ABB RAPID module: Module1.mod

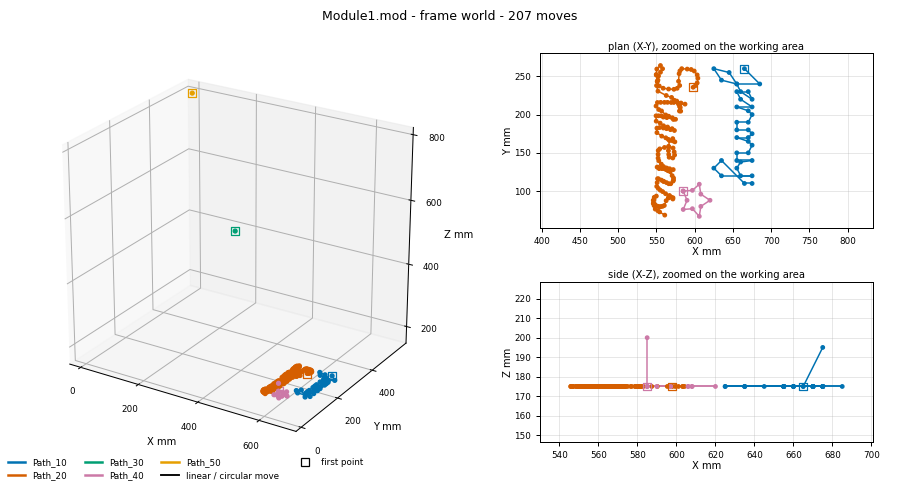
[picture p0: tool path of Module1.mod in frame world, 207 of 207 moves have a stored position in this frame; points joined in program order, loops and branches not executed]
MODULE Module1
    CONST robtarget Target_10:=[[45,210,0],[1,0,0,0],[0,0,-1,1],[9E+09,9E+09,9E+09,9E+09,9E+09,9E+09]];
    CONST robtarget Target_20:=[[25,190,0],[1,0,0,0],[0,0,-1,1],[9E+09,9E+09,9E+09,9E+09,9E+09,9E+09]];
    CONST robtarget Target_30:=[[55,190,0],[1,0,0,0],[0,0,-1,1],[9E+09,9E+09,9E+09,9E+09,9E+09,9E+09]];
    CONST robtarget Target_40:=[[75,195,0],[1,0,0,0],[0,0,-1,1],[9E+09,9E+09,9E+09,9E+09,9E+09,9E+09]];
    CONST robtarget Target_50:=[[85,210,0],[1,0,0,0],[0,0,-1,1],[9E+09,9E+09,9E+09,9E+09,9E+09,9E+09]];
    CONST robtarget Target_60:=[[65,205,0],[1,0,0,0],[0,0,-1,1],[9E+09,9E+09,9E+09,9E+09,9E+09,9E+09]];
    CONST robtarget Target_70:=[[55,190,0],[1,0,0,0],[0,0,-1,1],[9E+09,9E+09,9E+09,9E+09,9E+09,9E+09]];
    CONST robtarget Target_80:=[[50,180,0],[1,0,0,0],[0,0,-1,1],[9E+09,9E+09,9E+09,9E+09,9E+09,9E+09]];
    CONST robtarget Target_90:=[[35,170,0],[1,0,0,0],[0,0,-1,1],[9E+09,9E+09,9E+09,9E+09,9E+09,9E+09]];
    CONST robtarget Target_100:=[[40,180,0],[1,0,0,0],[0,0,-1,1],[9E+09,9E+09,9E+09,9E+09,9E+09,9E+09]];
    CONST robtarget Target_110:=[[55,180,0],[1,0,0,0],[0,0,-1,1],[9E+09,9E+09,9E+09,9E+09,9E+09,9E+09]];
    CONST robtarget Target_120:=[[50,170,0],[1,0,0,0],[0,0,-1,1],[9E+09,9E+09,9E+09,9E+09,9E+09,9E+09]];
    CONST robtarget Target_130:=[[35,160,0],[1,0,0,0],[0,0,-1,1],[9E+09,9E+09,9E+09,9E+09,9E+09,9E+09]];
    CONST robtarget Target_140:=[[55,160,0],[1,0,0,0],[0,0,-1,1],[9E+09,9E+09,9E+09,9E+09,9E+09,9E+09]];
    CONST robtarget Target_150:=[[40,155,0],[1,0,0,0],[0,0,-1,1],[9E+09,9E+09,9E+09,9E+09,9E+09,9E+09]];
    CONST robtarget Target_160:=[[35,150,0],[1,0,0,0],[0,0,-1,1],[9E+09,9E+09,9E+09,9E+09,9E+09,9E+09]];
    CONST robtarget Target_170:=[[40,140,0],[1,0,0,0],[0,0,-1,1],[9E+09,9E+09,9E+09,9E+09,9E+09,9E+09]];
    CONST robtarget Target_180:=[[55,140,0],[1,0,0,0],[0,0,-1,1],[9E+09,9E+09,9E+09,9E+09,9E+09,9E+09]];
    CONST robtarget Target_190:=[[55,130,0],[1,0,0,0],[0,0,-1,1],[9E+09,9E+09,9E+09,9E+09,9E+09,9E+09]];
    CONST robtarget Target_200:=[[40,130,0],[1,0,0,0],[0,0,-1,1],[9E+09,9E+09,9E+09,9E+09,9E+09,9E+09]];
    CONST robtarget Target_210:=[[35,125,0],[1,0,0,0],[0,0,-1,1],[9E+09,9E+09,9E+09,9E+09,9E+09,9E+09]];
    CONST robtarget Target_220:=[[40,120,0],[1,0,0,0],[0,0,-1,1],[9E+09,9E+09,9E+09,9E+09,9E+09,9E+09]];
    CONST robtarget Target_230:=[[55,120,0],[1,0,0,0],[0,0,-1,1],[9E+09,9E+09,9E+09,9E+09,9E+09,9E+09]];
    CONST robtarget Target_240:=[[40,115,0],[1,0,0,0],[0,0,-1,1],[9E+09,9E+09,9E+09,9E+09,9E+09,9E+09]];
    CONST robtarget Target_250:=[[35,110,0],[1,0,0,0],[0,0,-1,1],[9E+09,9E+09,9E+09,9E+09,9E+09,9E+09]];
    CONST robtarget Target_260:=[[40,100,0],[1,0,0,0],[0,0,-1,1],[9E+09,9E+09,9E+09,9E+09,9E+09,9E+09]];
    CONST robtarget Target_270:=[[55,100,0],[1,0,0,0],[0,0,-1,1],[9E+09,9E+09,9E+09,9E+09,9E+09,9E+09]];
    CONST robtarget Target_280:=[[55,90,0],[1,0,0,0],[0,0,-1,1],[9E+09,9E+09,9E+09,9E+09,9E+09,9E+09]];
    CONST robtarget Target_290:=[[35,90,0],[1,0,0,0],[0,0,-1,1],[9E+09,9E+09,9E+09,9E+09,9E+09,9E+09]];
    CONST robtarget Target_300:=[[50,88,0],[1,0,0,0],[0,0,-1,1],[9E+09,9E+09,9E+09,9E+09,9E+09,9E+09]];
    CONST robtarget Target_310:=[[55,80,0],[1,0,0,0],[0,0,-1,1],[9E+09,9E+09,9E+09,9E+09,9E+09,9E+09]];
    CONST robtarget Target_320:=[[50,70,0],[1,0,0,0],[0,0,-1,1],[9E+09,9E+09,9E+09,9E+09,9E+09,9E+09]];
    CONST robtarget Target_330:=[[35,70,0],[1,0,0,0],[0,0,-1,1],[9E+09,9E+09,9E+09,9E+09,9E+09,9E+09]];
    CONST robtarget Target_340:=[[75,70,0],[1,0,0,0],[0,0,-1,1],[9E+09,9E+09,9E+09,9E+09,9E+09,9E+09]];
    CONST robtarget Target_350:=[[85,80,0],[1,0,0,0],[0,0,-1,1],[9E+09,9E+09,9E+09,9E+09,9E+09,9E+09]];
    CONST robtarget Target_360:=[[75,90,0],[1,0,0,0],[0,0,-1,1],[9E+09,9E+09,9E+09,9E+09,9E+09,9E+09]];
    CONST robtarget Target_370:=[[45,60,0],[1,0,0,0],[0,0,-1,1],[9E+09,9E+09,9E+09,9E+09,9E+09,9E+09]];
    CONST robtarget Target_390:=[[108.942,187.897,0],[1,0,0,0],[0,0,-1,1],[9E+09,9E+09,9E+09,9E+09,9E+09,9E+09]];
    CONST robtarget Target_400:=[[106.749,191.385,0],[1,0,0,0],[0,0,-1,1],[9E+09,9E+09,9E+09,9E+09,9E+09,9E+09]];
    CONST robtarget Target_380:=[[112.054,185.689,0],[1,0,0,0],[0,0,-1,1],[9E+09,9E+09,9E+09,9E+09,9E+09,9E+09]];
    CONST robtarget Target_410:=[[105.843,197.618,0],[1,0,0,0],[0,0,-1,1],[9E+09,9E+09,9E+09,9E+09,9E+09,9E+09]];
    CONST robtarget Target_420:=[[106.766,201.829,0],[1,0,0,0],[0,0,-1,1],[9E+09,9E+09,9E+09,9E+09,9E+09,9E+09]];
    CONST robtarget Target_430:=[[110.623,206.946,0],[1,0,0,0],[0,0,-1,1],[9E+09,9E+09,9E+09,9E+09,9E+09,9E+09]];
    CONST robtarget Target_440:=[[114.657,208.948,0],[1,0,0,0],[0,0,-1,1],[9E+09,9E+09,9E+09,9E+09,9E+09,9E+09]];
    CONST robtarget Target_450:=[[119.787,209.479,0],[1,0,0,0],[0,0,-1,1],[9E+09,9E+09,9E+09,9E+09,9E+09,9E+09]];
    CONST robtarget Target_460:=[[126.931,210.004,0],[1,0,0,0],[0,0,-1,1],[9E+09,9E+09,9E+09,9E+09,9E+09,9E+09]];
    CONST robtarget Target_470:=[[129.306,207.065,0],[1,0,0,0],[0,0,-1,1],[9E+09,9E+09,9E+09,9E+09,9E+09,9E+09]];
    CONST robtarget Target_480:=[[130.399,203.399,0],[1,0,0,0],[0,0,-1,1],[9E+09,9E+09,9E+09,9E+09,9E+09,9E+09]];
    CONST robtarget Target_490:=[[131.115,193.507,0],[1,0,0,0],[0,0,-1,1],[9E+09,9E+09,9E+09,9E+09,9E+09,9E+09]];
    CONST robtarget Target_500:=[[129.641,188.017,0],[1,0,0,0],[0,0,-1,1],[9E+09,9E+09,9E+09,9E+09,9E+09,9E+09]];
    CONST robtarget Target_510:=[[132.931,184.344,0],[1,0,0,0],[0,0,-1,1],[9E+09,9E+09,9E+09,9E+09,9E+09,9E+09]];
    CONST robtarget Target_520:=[[137.139,183.05,0],[1,0,0,0],[0,0,-1,1],[9E+09,9E+09,9E+09,9E+09,9E+09,9E+09]];
    CONST robtarget Target_530:=[[144.094,183.396,0],[1,0,0,0],[0,0,-1,1],[9E+09,9E+09,9E+09,9E+09,9E+09,9E+09]];
    CONST robtarget Target_540:=[[151.231,184.473,0],[1,0,0,0],[0,0,-1,1],[9E+09,9E+09,9E+09,9E+09,9E+09,9E+09]];
    CONST robtarget Target_550:=[[156.358,187.386,0],[1,0,0,0],[0,0,-1,1],[9E+09,9E+09,9E+09,9E+09,9E+09,9E+09]];
    CONST robtarget Target_560:=[[158.928,193.236,0],[1,0,0,0],[0,0,-1,1],[9E+09,9E+09,9E+09,9E+09,9E+09,9E+09]];
    CONST robtarget Target_570:=[[158.929,193.602,0],[1,0,0,0],[0,0,-1,1],[9E+09,9E+09,9E+09,9E+09,9E+09,9E+09]];
    CONST robtarget Target_580:=[[160.222,201.651,0],[1,0,0,0],[0,0,-1,1],[9E+09,9E+09,9E+09,9E+09,9E+09,9E+09]];
    CONST robtarget Target_590:=[[160.223,202.383,0],[1,0,0,0],[0,0,-1,1],[9E+09,9E+09,9E+09,9E+09,9E+09,9E+09]];
    CONST robtarget Target_600:=[[159.504,209.524,0],[1,0,0,0],[0,0,-1,1],[9E+09,9E+09,9E+09,9E+09,9E+09,9E+09]];
    CONST robtarget Target_610:=[[154.756,214.117,0],[1,0,0,0],[0,0,-1,1],[9E+09,9E+09,9E+09,9E+09,9E+09,9E+09]];
    CONST robtarget Target_620:=[[152.005,209.916,0],[1,0,0,0],[0,0,-1,1],[9E+09,9E+09,9E+09,9E+09,9E+09,9E+09]];
    CONST robtarget Target_630:=[[154.741,205.33,0],[1,0,0,0],[0,0,-1,1],[9E+09,9E+09,9E+09,9E+09,9E+09,9E+09]];
    CONST robtarget Target_640:=[[157.294,200.379,0],[1,0,0,0],[0,0,-1,1],[9E+09,9E+09,9E+09,9E+09,9E+09,9E+09]];
    CONST robtarget Target_650:=[[158.017,195.069,0],[1,0,0,0],[0,0,-1,1],[9E+09,9E+09,9E+09,9E+09,9E+09,9E+09]];
    CONST robtarget Target_660:=[[159.834,187.925,0],[1,0,0,0],[0,0,-1,1],[9E+09,9E+09,9E+09,9E+09,9E+09,9E+09]];
    CONST robtarget Target_670:=[[157.993,180.609,0],[1,0,0,0],[0,0,-1,1],[9E+09,9E+09,9E+09,9E+09,9E+09,9E+09]];
    CONST robtarget Target_680:=[[147.191,174.965,0],[1,0,0,0],[0,0,-1,1],[9E+09,9E+09,9E+09,9E+09,9E+09,9E+09]];
    CONST robtarget Target_690:=[[140.233,172.421,0],[1,0,0,0],[0,0,-1,1],[9E+09,9E+09,9E+09,9E+09,9E+09,9E+09]];
    CONST robtarget Target_700:=[[136.749,168.768,0],[1,0,0,0],[0,0,-1,1],[9E+09,9E+09,9E+09,9E+09,9E+09,9E+09]];
    CONST robtarget Target_710:=[[133.452,167.678,0],[1,0,0,0],[0,0,-1,1],[9E+09,9E+09,9E+09,9E+09,9E+09,9E+09]];
    CONST robtarget Target_720:=[[127.955,165.128,0],[1,0,0,0],[0,0,-1,1],[9E+09,9E+09,9E+09,9E+09,9E+09,9E+09]];
    CONST robtarget Target_730:=[[122.642,163.677,0],[1,0,0,0],[0,0,-1,1],[9E+09,9E+09,9E+09,9E+09,9E+09,9E+09]];
    CONST robtarget Target_740:=[[128.504,164.578,0],[1,0,0,0],[0,0,-1,1],[9E+09,9E+09,9E+09,9E+09,9E+09,9E+09]];
    CONST robtarget Target_750:=[[129.779,160.545,0],[1,0,0,0],[0,0,-1,1],[9E+09,9E+09,9E+09,9E+09,9E+09,9E+09]];
    CONST robtarget Target_760:=[[129.952,154.684,0],[1,0,0,0],[0,0,-1,1],[9E+09,9E+09,9E+09,9E+09,9E+09,9E+09]];
    CONST robtarget Target_770:=[[128.304,154.505,0],[1,0,0,0],[0,0,-1,1],[9E+09,9E+09,9E+09,9E+09,9E+09,9E+09]];
    CONST robtarget Target_780:=[[128.861,159.265,0],[1,0,0,0],[0,0,-1,1],[9E+09,9E+09,9E+09,9E+09,9E+09,9E+09]];
    CONST robtarget Target_790:=[[131.249,163.838,0],[1,0,0,0],[0,0,-1,1],[9E+09,9E+09,9E+09,9E+09,9E+09,9E+09]];
    CONST robtarget Target_800:=[[137.293,165.837,0],[1,0,0,0],[0,0,-1,1],[9E+09,9E+09,9E+09,9E+09,9E+09,9E+09]];
    CONST robtarget Target_810:=[[140.771,165.828,0],[1,0,0,0],[0,0,-1,1],[9E+09,9E+09,9E+09,9E+09,9E+09,9E+09]];
    CONST robtarget Target_820:=[[145.529,165.998,0],[1,0,0,0],[0,0,-1,1],[9E+09,9E+09,9E+09,9E+09,9E+09,9E+09]];
    CONST robtarget Target_830:=[[149.554,165.988,0],[1,0,0,0],[0,0,-1,1],[9E+09,9E+09,9E+09,9E+09,9E+09,9E+09]];
    CONST robtarget Target_840:=[[154.494,165.975,0],[1,0,0,0],[0,0,-1,1],[9E+09,9E+09,9E+09,9E+09,9E+09,9E+09]];
    CONST robtarget Target_850:=[[158.7,165.781,0],[1,0,0,0],[0,0,-1,1],[9E+09,9E+09,9E+09,9E+09,9E+09,9E+09]];
    CONST robtarget Target_860:=[[160.521,161.2,0],[1,0,0,0],[0,0,-1,1],[9E+09,9E+09,9E+09,9E+09,9E+09,9E+09]];
    CONST robtarget Target_870:=[[157.039,156.633,0],[1,0,0,0],[0,0,-1,1],[9E+09,9E+09,9E+09,9E+09,9E+09,9E+09]];
    CONST robtarget Target_880:=[[153.378,154.811,0],[1,0,0,0],[0,0,-1,1],[9E+09,9E+09,9E+09,9E+09,9E+09,9E+09]];
    CONST robtarget Target_890:=[[147.881,149.515,0],[1,0,0,0],[0,0,-1,1],[9E+09,9E+09,9E+09,9E+09,9E+09,9E+09]];
    CONST robtarget Target_900:=[[144.035,147.876,0],[1,0,0,0],[0,0,-1,1],[9E+09,9E+09,9E+09,9E+09,9E+09,9E+09]];
    CONST robtarget Target_910:=[[139.274,145.873,0],[1,0,0,0],[0,0,-1,1],[9E+09,9E+09,9E+09,9E+09,9E+09,9E+09]];
    CONST robtarget Target_920:=[[135.061,143.868,0],[1,0,0,0],[0,0,-1,1],[9E+09,9E+09,9E+09,9E+09,9E+09,9E+09]];
    CONST robtarget Target_930:=[[137.806,143.679,0],[1,0,0,0],[0,0,-1,1],[9E+09,9E+09,9E+09,9E+09,9E+09,9E+09]];
    CONST robtarget Target_940:=[[146.411,146.04,0],[1,0,0,0],[0,0,-1,1],[9E+09,9E+09,9E+09,9E+09,9E+09,9E+09]];
    CONST robtarget Target_960:=[[153.733,148.403,0],[1,0,0,0],[0,0,-1,1],[9E+09,9E+09,9E+09,9E+09,9E+09,9E+09]];
    CONST robtarget Target_970:=[[157.391,148.395,0],[1,0,0,0],[0,0,-1,1],[9E+09,9E+09,9E+09,9E+09,9E+09,9E+09]];
    CONST robtarget Target_980:=[[160.5,148.388,0],[1,0,0,0],[0,0,-1,1],[9E+09,9E+09,9E+09,9E+09,9E+09,9E+09]];
    CONST robtarget Target_990:=[[160.306,141.433,0],[1,0,0,0],[0,0,-1,1],[9E+09,9E+09,9E+09,9E+09,9E+09,9E+09]];
    CONST robtarget Target_1000:=[[155.181,138.881,0],[1,0,0,0],[0,0,-1,1],[9E+09,9E+09,9E+09,9E+09,9E+09,9E+09]];
    CONST robtarget Target_1010:=[[150.785,135.412,0],[1,0,0,0],[0,0,-1,1],[9E+09,9E+09,9E+09,9E+09,9E+09,9E+09]];
    CONST robtarget Target_1020:=[[145.476,133.775,0],[1,0,0,0],[0,0,-1,1],[9E+09,9E+09,9E+09,9E+09,9E+09,9E+09]];
    CONST robtarget Target_1030:=[[139.616,131.59,0],[1,0,0,0],[0,0,-1,1],[9E+09,9E+09,9E+09,9E+09,9E+09,9E+09]];
    CONST robtarget Target_1040:=[[136.501,129.215,0],[1,0,0,0],[0,0,-1,1],[9E+09,9E+09,9E+09,9E+09,9E+09,9E+09]];
    CONST robtarget Target_1050:=[[141.627,130.304,0],[1,0,0,0],[0,0,-1,1],[9E+09,9E+09,9E+09,9E+09,9E+09,9E+09]];
    CONST robtarget Target_1060:=[[146.753,131.576,0],[1,0,0,0],[0,0,-1,1],[9E+09,9E+09,9E+09,9E+09,9E+09,9E+09]];
    CONST robtarget Target_1070:=[[150.963,132.483,0],[1,0,0,0],[0,0,-1,1],[9E+09,9E+09,9E+09,9E+09,9E+09,9E+09]];
    CONST robtarget Target_1080:=[[155.903,133.022,0],[1,0,0,0],[0,0,-1,1],[9E+09,9E+09,9E+09,9E+09,9E+09,9E+09]];
    CONST robtarget Target_1090:=[[159.376,132.284,0],[1,0,0,0],[0,0,-1,1],[9E+09,9E+09,9E+09,9E+09,9E+09,9E+09]];
    CONST robtarget Target_1100:=[[159.367,126.426,0],[1,0,0,0],[0,0,-1,1],[9E+09,9E+09,9E+09,9E+09,9E+09,9E+09]];
    CONST robtarget Target_1110:=[[153.14,121.861,0],[1,0,0,0],[0,0,-1,1],[9E+09,9E+09,9E+09,9E+09,9E+09,9E+09]];
    CONST robtarget Target_1120:=[[147.831,119.674,0],[1,0,0,0],[0,0,-1,1],[9E+09,9E+09,9E+09,9E+09,9E+09,9E+09]];
    CONST robtarget Target_1130:=[[144.535,117.665,0],[1,0,0,0],[0,0,-1,1],[9E+09,9E+09,9E+09,9E+09,9E+09,9E+09]];
    CONST robtarget Target_1140:=[[138.675,115.661,0],[1,0,0,0],[0,0,-1,1],[9E+09,9E+09,9E+09,9E+09,9E+09,9E+09]];
    CONST robtarget Target_1150:=[[135.927,114.383,0],[1,0,0,0],[0,0,-1,1],[9E+09,9E+09,9E+09,9E+09,9E+09,9E+09]];
    CONST robtarget Target_1160:=[[138.68,118.591,0],[1,0,0,0],[0,0,-1,1],[9E+09,9E+09,9E+09,9E+09,9E+09,9E+09]];
    CONST robtarget Target_1170:=[[142.885,116.02,0],[1,0,0,0],[0,0,-1,1],[9E+09,9E+09,9E+09,9E+09,9E+09,9E+09]];
    CONST robtarget Target_1180:=[[144.154,108.511,0],[1,0,0,0],[0,0,-1,1],[9E+09,9E+09,9E+09,9E+09,9E+09,9E+09]];
    CONST robtarget Target_1190:=[[144.327,102.835,0],[1,0,0,0],[0,0,-1,1],[9E+09,9E+09,9E+09,9E+09,9E+09,9E+09]];
    CONST robtarget Target_1200:=[[143.953,97.892,0],[1,0,0,0],[0,0,-1,1],[9E+09,9E+09,9E+09,9E+09,9E+09,9E+09]];
    CONST robtarget Target_1210:=[[143.398,94.231,0],[1,0,0,0],[0,0,-1,1],[9E+09,9E+09,9E+09,9E+09,9E+09,9E+09]];
    CONST robtarget Target_1220:=[[138.638,93.321,0],[1,0,0,0],[0,0,-1,1],[9E+09,9E+09,9E+09,9E+09,9E+09,9E+09]];
    CONST robtarget Target_1230:=[[136.265,97.17,0],[1,0,0,0],[0,0,-1,1],[9E+09,9E+09,9E+09,9E+09,9E+09,9E+09]];
    CONST robtarget Target_1240:=[[136.821,101.198,0],[1,0,0,0],[0,0,-1,1],[9E+09,9E+09,9E+09,9E+09,9E+09,9E+09]];
    CONST robtarget Target_1250:=[[138.294,106.323,0],[1,0,0,0],[0,0,-1,1],[9E+09,9E+09,9E+09,9E+09,9E+09,9E+09]];
    CONST robtarget Target_1260:=[[143.786,107.597,0],[1,0,0,0],[0,0,-1,1],[9E+09,9E+09,9E+09,9E+09,9E+09,9E+09]];
    CONST robtarget Target_1270:=[[149.457,107.039,0],[1,0,0,0],[0,0,-1,1],[9E+09,9E+09,9E+09,9E+09,9E+09,9E+09]];
    CONST robtarget Target_1280:=[[155.674,105.2,0],[1,0,0,0],[0,0,-1,1],[9E+09,9E+09,9E+09,9E+09,9E+09,9E+09]];
    CONST robtarget Target_1290:=[[157.682,103,0],[1,0,0,0],[0,0,-1,1],[9E+09,9E+09,9E+09,9E+09,9E+09,9E+09]];
    CONST robtarget Target_1300:=[[157.857,98.058,0],[1,0,0,0],[0,0,-1,1],[9E+09,9E+09,9E+09,9E+09,9E+09,9E+09]];
    CONST robtarget Target_1310:=[[157.849,93.116,0],[1,0,0,0],[0,0,-1,1],[9E+09,9E+09,9E+09,9E+09,9E+09,9E+09]];
    CONST robtarget Target_1320:=[[156.928,89.639,0],[1,0,0,0],[0,0,-1,1],[9E+09,9E+09,9E+09,9E+09,9E+09,9E+09]];
    CONST robtarget Target_1330:=[[153.629,85.25,0],[1,0,0,0],[0,0,-1,1],[9E+09,9E+09,9E+09,9E+09,9E+09,9E+09]];
    CONST robtarget Target_1340:=[[150.88,82.14,0],[1,0,0,0],[0,0,-1,1],[9E+09,9E+09,9E+09,9E+09,9E+09,9E+09]];
    CONST robtarget Target_1350:=[[147.035,80.313,0],[1,0,0,0],[0,0,-1,1],[9E+09,9E+09,9E+09,9E+09,9E+09,9E+09]];
    CONST robtarget Target_1360:=[[142.824,79.218,0],[1,0,0,0],[0,0,-1,1],[9E+09,9E+09,9E+09,9E+09,9E+09,9E+09]];
    CONST robtarget Target_1370:=[[138.064,78.124,0],[1,0,0,0],[0,0,-1,1],[9E+09,9E+09,9E+09,9E+09,9E+09,9E+09]];
    CONST robtarget Target_1380:=[[141.907,77.754,0],[1,0,0,0],[0,0,-1,1],[9E+09,9E+09,9E+09,9E+09,9E+09,9E+09]];
    CONST robtarget Target_1390:=[[145.752,79.216,0],[1,0,0,0],[0,0,-1,1],[9E+09,9E+09,9E+09,9E+09,9E+09,9E+09]];
    CONST robtarget Target_1400:=[[149.412,79.396,0],[1,0,0,0],[0,0,-1,1],[9E+09,9E+09,9E+09,9E+09,9E+09,9E+09]];
    CONST robtarget Target_1410:=[[154.17,80.856,0],[1,0,0,0],[0,0,-1,1],[9E+09,9E+09,9E+09,9E+09,9E+09,9E+09]];
    CONST robtarget Target_1420:=[[158.012,81.218,0],[1,0,0,0],[0,0,-1,1],[9E+09,9E+09,9E+09,9E+09,9E+09,9E+09]];
    CONST robtarget Target_1430:=[[159.11,81.4,0],[1,0,0,0],[0,0,-1,1],[9E+09,9E+09,9E+09,9E+09,9E+09,9E+09]];
    CONST robtarget Target_1440:=[[156.546,79.389,0],[1,0,0,0],[0,0,-1,1],[9E+09,9E+09,9E+09,9E+09,9E+09,9E+09]];
    CONST robtarget Target_1450:=[[152.888,79.392,0],[1,0,0,0],[0,0,-1,1],[9E+09,9E+09,9E+09,9E+09,9E+09,9E+09]];
    CONST robtarget Target_1460:=[[150.327,79.578,0],[1,0,0,0],[0,0,-1,1],[9E+09,9E+09,9E+09,9E+09,9E+09,9E+09]];
    CONST robtarget Target_1470:=[[147.58,78.116,0],[1,0,0,0],[0,0,-1,1],[9E+09,9E+09,9E+09,9E+09,9E+09,9E+09]];
    CONST robtarget Target_1480:=[[145.016,76.653,0],[1,0,0,0],[0,0,-1,1],[9E+09,9E+09,9E+09,9E+09,9E+09,9E+09]];
    CONST robtarget Target_1490:=[[142.086,75.374,0],[1,0,0,0],[0,0,-1,1],[9E+09,9E+09,9E+09,9E+09,9E+09,9E+09]];
    CONST robtarget Target_1500:=[[139.515,70.249,0],[1,0,0,0],[0,0,-1,1],[9E+09,9E+09,9E+09,9E+09,9E+09,9E+09]];
    CONST robtarget Target_1510:=[[137.68,67.137,0],[1,0,0,0],[0,0,-1,1],[9E+09,9E+09,9E+09,9E+09,9E+09,9E+09]];
    CONST robtarget Target_1520:=[[137.676,64.574,0],[1,0,0,0],[0,0,-1,1],[9E+09,9E+09,9E+09,9E+09,9E+09,9E+09]];
    CONST robtarget Target_1530:=[[138.222,63.109,0],[1,0,0,0],[0,0,-1,1],[9E+09,9E+09,9E+09,9E+09,9E+09,9E+09]];
    CONST robtarget Target_1540:=[[141.328,59.628,0],[1,0,0,0],[0,0,-1,1],[9E+09,9E+09,9E+09,9E+09,9E+09,9E+09]];
    CONST robtarget Target_1550:=[[143.89,59.627,0],[1,0,0,0],[0,0,-1,1],[9E+09,9E+09,9E+09,9E+09,9E+09,9E+09]];
    CONST robtarget Target_1560:=[[146.82,61.09,0],[1,0,0,0],[0,0,-1,1],[9E+09,9E+09,9E+09,9E+09,9E+09,9E+09]];
    CONST robtarget Target_1570:=[[150.299,62.553,0],[1,0,0,0],[0,0,-1,1],[9E+09,9E+09,9E+09,9E+09,9E+09,9E+09]];
    CONST robtarget Target_1580:=[[151.031,62.918,0],[1,0,0,0],[0,0,-1,1],[9E+09,9E+09,9E+09,9E+09,9E+09,9E+09]];
    CONST robtarget Target_1590:=[[153.594,64.381,0],[1,0,0,0],[0,0,-1,1],[9E+09,9E+09,9E+09,9E+09,9E+09,9E+09]];
    CONST robtarget Target_1600:=[[157.255,66.026,0],[1,0,0,0],[0,0,-1,1],[9E+09,9E+09,9E+09,9E+09,9E+09,9E+09]];
    CONST robtarget Target_1610:=[[158.536,66.209,0],[1,0,0,0],[0,0,-1,1],[9E+09,9E+09,9E+09,9E+09,9E+09,9E+09]];
    CONST robtarget Target_1620:=[[159.076,61.083,0],[1,0,0,0],[0,0,-1,1],[9E+09,9E+09,9E+09,9E+09,9E+09,9E+09]];
    CONST robtarget Target_1630:=[[159.617,56.141,0],[1,0,0,0],[0,0,-1,1],[9E+09,9E+09,9E+09,9E+09,9E+09,9E+09]];
    CONST robtarget Target_1640:=[[157.601,53.58,0],[1,0,0,0],[0,0,-1,1],[9E+09,9E+09,9E+09,9E+09,9E+09,9E+09]];
    CONST robtarget Target_1650:=[[155.036,51.201,0],[1,0,0,0],[0,0,-1,1],[9E+09,9E+09,9E+09,9E+09,9E+09,9E+09]];
    CONST robtarget Target_1660:=[[151.923,49.371,0],[1,0,0,0],[0,0,-1,1],[9E+09,9E+09,9E+09,9E+09,9E+09,9E+09]];
    CONST robtarget Target_1670:=[[148.077,46.626,0],[1,0,0,0],[0,0,-1,1],[9E+09,9E+09,9E+09,9E+09,9E+09,9E+09]];
    CONST robtarget Target_1680:=[[142.95,44.247,0],[1,0,0,0],[0,0,-1,1],[9E+09,9E+09,9E+09,9E+09,9E+09,9E+09]];
    CONST robtarget Target_1690:=[[138.55,39.67,0],[1,0,0,0],[0,0,-1,1],[9E+09,9E+09,9E+09,9E+09,9E+09,9E+09]];
    CONST robtarget Target_1700:=[[138.369,41.318,0],[1,0,0,0],[0,0,-1,1],[9E+09,9E+09,9E+09,9E+09,9E+09,9E+09]];
    CONST robtarget Target_1710:=[[140.567,42.05,0],[1,0,0,0],[0,0,-1,1],[9E+09,9E+09,9E+09,9E+09,9E+09,9E+09]];
    CONST robtarget Target_1720:=[[143.13,42.599,0],[1,0,0,0],[0,0,-1,1],[9E+09,9E+09,9E+09,9E+09,9E+09,9E+09]];
    CONST robtarget Target_1730:=[[144.226,41.501,0],[1,0,0,0],[0,0,-1,1],[9E+09,9E+09,9E+09,9E+09,9E+09,9E+09]];
    CONST robtarget Target_1740:=[[144.408,40.951,0],[1,0,0,0],[0,0,-1,1],[9E+09,9E+09,9E+09,9E+09,9E+09,9E+09]];
    CONST robtarget Target_1750:=[[147.33,37.473,0],[1,0,0,0],[0,0,-1,1],[9E+09,9E+09,9E+09,9E+09,9E+09,9E+09]];
    CONST robtarget Target_1760:=[[149.698,31.248,0],[1,0,0,0],[0,0,-1,1],[9E+09,9E+09,9E+09,9E+09,9E+09,9E+09]];
    CONST robtarget Target_1770:=[[151.892,30.15,0],[1,0,0,0],[0,0,-1,1],[9E+09,9E+09,9E+09,9E+09,9E+09,9E+09]];
    CONST robtarget Target_1780:=[[154.086,29.784,0],[1,0,0,0],[0,0,-1,1],[9E+09,9E+09,9E+09,9E+09,9E+09,9E+09]];
    CONST robtarget Target_1790:=[[156.098,29.601,0],[1,0,0,0],[0,0,-1,1],[9E+09,9E+09,9E+09,9E+09,9E+09,9E+09]];
    CONST robtarget Target_1800:=[[158.111,30.15,0],[1,0,0,0],[0,0,-1,1],[9E+09,9E+09,9E+09,9E+09,9E+09,9E+09]];
    CONST robtarget Target_1810:=[[161.405,31.981,0],[1,0,0,0],[0,0,-1,1],[9E+09,9E+09,9E+09,9E+09,9E+09,9E+09]];
    CONST robtarget Target_1820:=[[164.151,33.811,0],[1,0,0,0],[0,0,-1,1],[9E+09,9E+09,9E+09,9E+09,9E+09,9E+09]];
    CONST robtarget Target_1830:=[[164.158,37.838,0],[1,0,0,0],[0,0,-1,1],[9E+09,9E+09,9E+09,9E+09,9E+09,9E+09]];
    CONST robtarget Target_1840:=[[162.885,41.864,0],[1,0,0,0],[0,0,-1,1],[9E+09,9E+09,9E+09,9E+09,9E+09,9E+09]];
    CONST robtarget Target_1850:=[[160.144,43.512,0],[1,0,0,0],[0,0,-1,1],[9E+09,9E+09,9E+09,9E+09,9E+09,9E+09]];
    CONST robtarget Target_1860:=[[163.245,38.753,0],[1,0,0,0],[0,0,-1,1],[9E+09,9E+09,9E+09,9E+09,9E+09,9E+09]];
    CONST robtarget Target_1870:=[[163.604,34.543,0],[1,0,0,0],[0,0,-1,1],[9E+09,9E+09,9E+09,9E+09,9E+09,9E+09]];
    CONST robtarget Target_1880:=[[163.05,31.066,0],[1,0,0,0],[0,0,-1,1],[9E+09,9E+09,9E+09,9E+09,9E+09,9E+09]];
    CONST robtarget Target_1890:=[[161.579,26.49,0],[1,0,0,0],[0,0,-1,1],[9E+09,9E+09,9E+09,9E+09,9E+09,9E+09]];
    CONST robtarget Target_1900:=[[158.101,24.293,0],[1,0,0,0],[0,0,-1,1],[9E+09,9E+09,9E+09,9E+09,9E+09,9E+09]];
    CONST robtarget Target_1910:=[[155.904,22.828,0],[1,0,0,0],[0,0,-1,1],[9E+09,9E+09,9E+09,9E+09,9E+09,9E+09]];
    CONST robtarget Target_1920:=[[149.128,18.616,0],[1,0,0,0],[0,0,-1,1],[9E+09,9E+09,9E+09,9E+09,9E+09,9E+09]];
    CONST robtarget Target_950:=[[150.986,146.762,0],[1,0,0,0],[0,0,-1,1],[9E+09,9E+09,9E+09,9E+09,9E+09,9E+09]];
    CONST robtarget Target_Home:=[[506.291651246,0,679.5],[0.5,0,0.866025404,0],[0,0,-1,1],[9E+09,9E+09,9E+09,9E+09,9E+09,9E+09]];
    CONST robtarget Target_Up_first:=[[35,60,-20],[1,0,0,0],[0,0,-1,1],[9E+09,9E+09,9E+09,9E+09,9E+09,9E+09]];
    CONST robtarget Target_1930:=[[125,50,0],[1,0,0,0],[0,0,-1,1],[9E+09,9E+09,9E+09,9E+09,9E+09,9E+09]];
    CONST robtarget Target_1940:=[[120,38,0],[1,0,0,0],[0,0,-1,1],[9E+09,9E+09,9E+09,9E+09,9E+09,9E+09]];
    CONST robtarget Target_1950:=[[125,26,0],[1,0,0,0],[0,0,-1,1],[9E+09,9E+09,9E+09,9E+09,9E+09,9E+09]];
    CONST robtarget Target_1960:=[[113,27,0],[1,0,0,0],[0,0,-1,1],[9E+09,9E+09,9E+09,9E+09,9E+09,9E+09]];
    CONST robtarget Target_1970:=[[104,17,0],[1,0,0,0],[0,0,-1,1],[9E+09,9E+09,9E+09,9E+09,9E+09,9E+09]];
    CONST robtarget Target_1980:=[[102,30,0],[1,0,0,0],[0,0,-1,1],[9E+09,9E+09,9E+09,9E+09,9E+09,9E+09]];
    CONST robtarget Target_1990:=[[90,38,0],[1,0,0,0],[0,0,-1,1],[9E+09,9E+09,9E+09,9E+09,9E+09,9E+09]];
    CONST robtarget Target_2000:=[[102,46,0],[1,0,0,0],[0,0,-1,1],[9E+09,9E+09,9E+09,9E+09,9E+09,9E+09]];
    CONST robtarget Target_2010:=[[104,59,0],[1,0,0,0],[0,0,-1,1],[9E+09,9E+09,9E+09,9E+09,9E+09,9E+09]];
    CONST robtarget Target_2020:=[[113,51,0],[1,0,0,0],[0,0,-1,1],[9E+09,9E+09,9E+09,9E+09,9E+09,9E+09]];
    CONST robtarget Target_2040:=[[125,50,-25],[1,0,0,0],[0,0,-1,1],[9E+09,9E+09,9E+09,9E+09,9E+09,9E+09]];
    CONST robtarget Target_2080:=[[-21.410821192,47.500000043,-189.127099576],[0.991882579,0,0.127157185,0],[0,-1,0,0],[9E+09,9E+09,9E+09,9E+09,9E+09,9E+09]];
    CONST robtarget Target_2070:=[[27.859035711,47.500000049,-268.869437494],[0.996403223,0,0.084738521,0],[0,-1,0,0],[9E+09,9E+09,9E+09,9E+09,9E+09,9E+09]];
    CONST robtarget Target_2090:=[[44.999981721,209.999999917,0.000013697],[1,-0.000000001,-0.000000007,-0.000000008],[0,0,-1,1],[9E+09,9E+09,9E+09,9E+09,9E+09,9E+09]];
    CONST robtarget Target_2050:=[[715.334377905,668.594248012,-598.20561877],[0.629441784,-0.317048898,-0.313611408,-0.636341827],[1,1,-3,0],[9E+09,9E+09,9E+09,9E+09,9E+09,9E+09]];
    CONST robtarget Target_2060:=[[-6.301731189,578.000166138,792.762334881],[0.586316286,-0.392563698,0.388306911,0.592743366],[1,2,-3,0],[9E+09,9E+09,9E+09,9E+09,9E+09,9E+09]];
    PERS tooldata Marcador_R:=[TRUE,[[72.862,-2.5,121.799],[0.866025404,0,0.5,0]],[1,[0,0,1],[1,0,0,0],0,0,0]];
    TASK PERS wobjdata Wo_Caja:=[FALSE,TRUE,"",[[710,50,175],[0,0,1,0]],[[0,0,0],[1,0,0,0]]];


    PROC main()
        Path_30;
        WHILE TRUE DO
            IF DI_01 = 1 THEN
                Set DO_01;
                Path_30;
                Path_10;
                Path_40;
                Path_20;
                Path_30;
                Set DO_02;
                WaitTime 5.0;
                Reset DO_02;
            ENDIF
            IF DI_02=1 THEN
                Reset DO_01;
                Path_50;
            ENDIF
        ENDWHILE

    ENDPROC
    PROC Path_10()


        MoveJ Target_10,v100,z10,Marcador_R\WObj:=Wo_Caja;
        MoveL Target_20,v100,z10,Marcador_R\WObj:=Wo_Caja;
        MoveL Target_30,v100,z10,Marcador_R\WObj:=Wo_Caja;
        MoveL Target_40,v100,z10,Marcador_R\WObj:=Wo_Caja;
        MoveL Target_50,v100,z10,Marcador_R\WObj:=Wo_Caja;
        MoveL Target_60,v100,z10,Marcador_R\WObj:=Wo_Caja;
        MoveL Target_70,v100,z10,Marcador_R\WObj:=Wo_Caja;
        MoveL Target_80,v100,z10,Marcador_R\WObj:=Wo_Caja;
        MoveL Target_90,v100,z10,Marcador_R\WObj:=Wo_Caja;
        MoveL Target_100,v100,z10,Marcador_R\WObj:=Wo_Caja;
        MoveL Target_110,v100,z10,Marcador_R\WObj:=Wo_Caja;
        MoveL Target_120,v100,z10,Marcador_R\WObj:=Wo_Caja;
        MoveL Target_130,v100,z10,Marcador_R\WObj:=Wo_Caja;
        MoveL Target_140,v100,z10,Marcador_R\WObj:=Wo_Caja;
        MoveL Target_150,v100,z10,Marcador_R\WObj:=Wo_Caja;
        MoveL Target_160,v100,z10,Marcador_R\WObj:=Wo_Caja;
        MoveL Target_170,v100,z10,Marcador_R\WObj:=Wo_Caja;
        MoveL Target_180,v100,z10,Marcador_R\WObj:=Wo_Caja;
        MoveL Target_190,v100,z10,Marcador_R\WObj:=Wo_Caja;
        MoveL Target_200,v100,z10,Marcador_R\WObj:=Wo_Caja;
        MoveL Target_210,v100,z10,Marcador_R\WObj:=Wo_Caja;
        MoveL Target_220,v100,z10,Marcador_R\WObj:=Wo_Caja;
        MoveL Target_230,v100,z10,Marcador_R\WObj:=Wo_Caja;
        MoveL Target_240,v100,z10,Marcador_R\WObj:=Wo_Caja;
        MoveL Target_250,v100,z10,Marcador_R\WObj:=Wo_Caja;
        MoveL Target_260,v100,z10,Marcador_R\WObj:=Wo_Caja;
        MoveL Target_270,v100,z10,Marcador_R\WObj:=Wo_Caja;
        MoveL Target_280,v100,z10,Marcador_R\WObj:=Wo_Caja;
        MoveL Target_290,v100,z10,Marcador_R\WObj:=Wo_Caja;
        MoveL Target_300,v100,z10,Marcador_R\WObj:=Wo_Caja;
        MoveL Target_310,v100,z10,Marcador_R\WObj:=Wo_Caja;
        MoveL Target_320,v100,z10,Marcador_R\WObj:=Wo_Caja;
        MoveL Target_330,v100,z10,Marcador_R\WObj:=Wo_Caja;
        MoveL Target_340,v100,z10,Marcador_R\WObj:=Wo_Caja;
        MoveL Target_350,v100,z10,Marcador_R\WObj:=Wo_Caja;
        MoveL Target_360,v100,z10,Marcador_R\WObj:=Wo_Caja;
        MoveL Target_370,v100,z10,Marcador_R\WObj:=Wo_Caja;
        MoveL Target_Up_first,v1000,z100,Marcador_R\WObj:=Wo_Caja;
    ENDPROC
    PROC Path_20()
        MoveJ Target_380,v100,z10,Marcador_R\WObj:=Wo_Caja;
        MoveL Target_390,v100,z10,Marcador_R\WObj:=Wo_Caja;
        MoveL Target_400,v100,z10,Marcador_R\WObj:=Wo_Caja;
        MoveL Target_410,v100,z10,Marcador_R\WObj:=Wo_Caja;
        MoveL Target_420,v100,z10,Marcador_R\WObj:=Wo_Caja;
        MoveL Target_430,v100,z10,Marcador_R\WObj:=Wo_Caja;
        MoveL Target_440,v100,z10,Marcador_R\WObj:=Wo_Caja;
        MoveL Target_450,v100,z10,Marcador_R\WObj:=Wo_Caja;
        MoveL Target_460,v100,z10,Marcador_R\WObj:=Wo_Caja;
        MoveL Target_470,v100,z10,Marcador_R\WObj:=Wo_Caja;
        MoveL Target_480,v100,z10,Marcador_R\WObj:=Wo_Caja;
        MoveL Target_490,v100,z10,Marcador_R\WObj:=Wo_Caja;
        MoveL Target_500,v100,z10,Marcador_R\WObj:=Wo_Caja;
        MoveL Target_510,v100,z10,Marcador_R\WObj:=Wo_Caja;
        MoveL Target_520,v100,z10,Marcador_R\WObj:=Wo_Caja;
        MoveL Target_530,v100,z10,Marcador_R\WObj:=Wo_Caja;
        MoveL Target_540,v100,z10,Marcador_R\WObj:=Wo_Caja;
        MoveL Target_550,v100,z10,Marcador_R\WObj:=Wo_Caja;
        MoveL Target_560,v100,z10,Marcador_R\WObj:=Wo_Caja;
        MoveL Target_570,v100,z10,Marcador_R\WObj:=Wo_Caja;
        MoveL Target_580,v100,z10,Marcador_R\WObj:=Wo_Caja;
        MoveL Target_590,v100,z10,Marcador_R\WObj:=Wo_Caja;
        MoveL Target_600,v100,z10,Marcador_R\WObj:=Wo_Caja;
        MoveL Target_610,v100,z10,Marcador_R\WObj:=Wo_Caja;
        MoveL Target_620,v100,z10,Marcador_R\WObj:=Wo_Caja;
        MoveL Target_630,v100,z10,Marcador_R\WObj:=Wo_Caja;
        MoveL Target_640,v100,z10,Marcador_R\WObj:=Wo_Caja;
        MoveL Target_650,v100,z10,Marcador_R\WObj:=Wo_Caja;
        MoveL Target_660,v100,z10,Marcador_R\WObj:=Wo_Caja;
        MoveL Target_670,v100,z10,Marcador_R\WObj:=Wo_Caja;
        MoveL Target_680,v100,z10,Marcador_R\WObj:=Wo_Caja;
        MoveL Target_690,v100,z10,Marcador_R\WObj:=Wo_Caja;
        MoveL Target_700,v100,z10,Marcador_R\WObj:=Wo_Caja;
        MoveL Target_710,v100,z10,Marcador_R\WObj:=Wo_Caja;
        MoveL Target_720,v100,z10,Marcador_R\WObj:=Wo_Caja;
        MoveL Target_730,v100,z10,Marcador_R\WObj:=Wo_Caja;
        MoveL Target_740,v100,z10,Marcador_R\WObj:=Wo_Caja;
        MoveL Target_750,v100,z10,Marcador_R\WObj:=Wo_Caja;
        MoveL Target_760,v100,z10,Marcador_R\WObj:=Wo_Caja;
        MoveL Target_770,v100,z10,Marcador_R\WObj:=Wo_Caja;
        MoveL Target_780,v100,z10,Marcador_R\WObj:=Wo_Caja;
        MoveL Target_790,v100,z10,Marcador_R\WObj:=Wo_Caja;
        MoveL Target_800,v100,z10,Marcador_R\WObj:=Wo_Caja;
        MoveL Target_810,v100,z10,Marcador_R\WObj:=Wo_Caja;
        MoveL Target_820,v100,z10,Marcador_R\WObj:=Wo_Caja;
        MoveL Target_830,v100,z10,Marcador_R\WObj:=Wo_Caja;
        MoveL Target_840,v100,z10,Marcador_R\WObj:=Wo_Caja;
        MoveL Target_850,v100,z10,Marcador_R\WObj:=Wo_Caja;
        MoveL Target_860,v100,z10,Marcador_R\WObj:=Wo_Caja;
        MoveL Target_870,v100,z10,Marcador_R\WObj:=Wo_Caja;
        MoveL Target_880,v100,z10,Marcador_R\WObj:=Wo_Caja;
        MoveL Target_890,v100,z10,Marcador_R\WObj:=Wo_Caja;
        MoveL Target_900,v100,z10,Marcador_R\WObj:=Wo_Caja;
        MoveL Target_910,v100,z10,Marcador_R\WObj:=Wo_Caja;
        MoveL Target_920,v100,z10,Marcador_R\WObj:=Wo_Caja;
        MoveL Target_930,v100,z10,Marcador_R\WObj:=Wo_Caja;
        MoveL Target_940,v100,z10,Marcador_R\WObj:=Wo_Caja;
        MoveL Target_950,v100,z10,Marcador_R\WObj:=Wo_Caja;
        MoveL Target_960,v100,z10,Marcador_R\WObj:=Wo_Caja;
        MoveL Target_970,v100,z10,Marcador_R\WObj:=Wo_Caja;
        MoveL Target_980,v100,z10,Marcador_R\WObj:=Wo_Caja;
        MoveL Target_990,v100,z10,Marcador_R\WObj:=Wo_Caja;
        MoveL Target_1000,v100,z10,Marcador_R\WObj:=Wo_Caja;
        MoveL Target_1010,v100,z10,Marcador_R\WObj:=Wo_Caja;
        MoveL Target_1020,v100,z10,Marcador_R\WObj:=Wo_Caja;
        MoveL Target_1030,v100,z10,Marcador_R\WObj:=Wo_Caja;
        MoveL Target_1040,v100,z10,Marcador_R\WObj:=Wo_Caja;
        MoveL Target_1050,v100,z10,Marcador_R\WObj:=Wo_Caja;
        MoveL Target_1060,v100,z10,Marcador_R\WObj:=Wo_Caja;
        MoveL Target_1070,v100,z10,Marcador_R\WObj:=Wo_Caja;
        MoveL Target_1080,v100,z10,Marcador_R\WObj:=Wo_Caja;
        MoveL Target_1090,v100,z10,Marcador_R\WObj:=Wo_Caja;
        MoveL Target_1100,v100,z10,Marcador_R\WObj:=Wo_Caja;
        MoveL Target_1110,v100,z10,Marcador_R\WObj:=Wo_Caja;
        MoveL Target_1120,v100,z10,Marcador_R\WObj:=Wo_Caja;
        MoveL Target_1130,v100,z10,Marcador_R\WObj:=Wo_Caja;
        MoveL Target_1140,v100,z10,Marcador_R\WObj:=Wo_Caja;
        MoveL Target_1150,v100,z10,Marcador_R\WObj:=Wo_Caja;
        MoveL Target_1160,v100,z10,Marcador_R\WObj:=Wo_Caja;
        MoveL Target_1170,v100,z10,Marcador_R\WObj:=Wo_Caja;
        MoveL Target_1180,v100,z10,Marcador_R\WObj:=Wo_Caja;
        MoveL Target_1190,v100,z10,Marcador_R\WObj:=Wo_Caja;
        MoveL Target_1200,v100,z10,Marcador_R\WObj:=Wo_Caja;
        MoveL Target_1210,v100,z10,Marcador_R\WObj:=Wo_Caja;
        MoveL Target_1220,v100,z10,Marcador_R\WObj:=Wo_Caja;
        MoveL Target_1230,v100,z10,Marcador_R\WObj:=Wo_Caja;
        MoveL Target_1240,v100,z10,Marcador_R\WObj:=Wo_Caja;
        MoveL Target_1250,v100,z10,Marcador_R\WObj:=Wo_Caja;
        MoveL Target_1260,v100,z10,Marcador_R\WObj:=Wo_Caja;
        MoveL Target_1270,v100,z10,Marcador_R\WObj:=Wo_Caja;
        MoveL Target_1280,v100,z10,Marcador_R\WObj:=Wo_Caja;
        MoveL Target_1290,v100,z10,Marcador_R\WObj:=Wo_Caja;
        MoveL Target_1300,v100,z10,Marcador_R\WObj:=Wo_Caja;
        MoveL Target_1310,v100,z10,Marcador_R\WObj:=Wo_Caja;
        MoveL Target_1320,v100,z10,Marcador_R\WObj:=Wo_Caja;
        MoveL Target_1330,v100,z10,Marcador_R\WObj:=Wo_Caja;
        MoveL Target_1340,v100,z10,Marcador_R\WObj:=Wo_Caja;
        MoveL Target_1350,v100,z10,Marcador_R\WObj:=Wo_Caja;
        MoveL Target_1360,v100,z10,Marcador_R\WObj:=Wo_Caja;
        MoveL Target_1370,v100,z10,Marcador_R\WObj:=Wo_Caja;
        MoveL Target_1380,v100,z10,Marcador_R\WObj:=Wo_Caja;
        MoveL Target_1390,v100,z10,Marcador_R\WObj:=Wo_Caja;
        MoveL Target_1400,v100,z10,Marcador_R\WObj:=Wo_Caja;
        MoveL Target_1410,v100,z10,Marcador_R\WObj:=Wo_Caja;
        MoveL Target_1420,v100,z10,Marcador_R\WObj:=Wo_Caja;
        MoveL Target_1430,v100,z10,Marcador_R\WObj:=Wo_Caja;
        MoveL Target_1440,v100,z10,Marcador_R\WObj:=Wo_Caja;
        MoveL Target_1450,v100,z10,Marcador_R\WObj:=Wo_Caja;
        MoveL Target_1460,v100,z10,Marcador_R\WObj:=Wo_Caja;
        MoveL Target_1470,v100,z10,Marcador_R\WObj:=Wo_Caja;
        MoveL Target_1480,v100,z10,Marcador_R\WObj:=Wo_Caja;
        MoveL Target_1490,v100,z10,Marcador_R\WObj:=Wo_Caja;
        MoveL Target_1500,v100,z10,Marcador_R\WObj:=Wo_Caja;
        MoveL Target_1510,v100,z10,Marcador_R\WObj:=Wo_Caja;
        MoveL Target_1520,v100,z10,Marcador_R\WObj:=Wo_Caja;
        MoveL Target_1530,v100,z10,Marcador_R\WObj:=Wo_Caja;
        MoveL Target_1540,v100,z10,Marcador_R\WObj:=Wo_Caja;
        MoveL Target_1550,v100,z10,Marcador_R\WObj:=Wo_Caja;
        MoveL Target_1560,v100,z10,Marcador_R\WObj:=Wo_Caja;
        MoveL Target_1570,v100,z10,Marcador_R\WObj:=Wo_Caja;
        MoveL Target_1580,v100,z10,Marcador_R\WObj:=Wo_Caja;
        MoveL Target_1590,v100,z10,Marcador_R\WObj:=Wo_Caja;
        MoveL Target_1600,v100,z10,Marcador_R\WObj:=Wo_Caja;
        MoveL Target_1610,v100,z10,Marcador_R\WObj:=Wo_Caja;
        MoveL Target_1620,v100,z10,Marcador_R\WObj:=Wo_Caja;
        MoveL Target_1630,v100,z10,Marcador_R\WObj:=Wo_Caja;
        MoveL Target_1640,v100,z10,Marcador_R\WObj:=Wo_Caja;
        MoveL Target_1650,v100,z10,Marcador_R\WObj:=Wo_Caja;
        MoveL Target_1660,v100,z10,Marcador_R\WObj:=Wo_Caja;
        MoveL Target_1670,v100,z10,Marcador_R\WObj:=Wo_Caja;
        MoveL Target_1680,v100,z10,Marcador_R\WObj:=Wo_Caja;
        MoveL Target_1690,v100,z10,Marcador_R\WObj:=Wo_Caja;
        MoveL Target_1700,v100,z10,Marcador_R\WObj:=Wo_Caja;
        MoveL Target_1710,v100,z10,Marcador_R\WObj:=Wo_Caja;
        MoveL Target_1720,v100,z10,Marcador_R\WObj:=Wo_Caja;
        MoveL Target_1730,v100,z10,Marcador_R\WObj:=Wo_Caja;
        MoveL Target_1740,v100,z10,Marcador_R\WObj:=Wo_Caja;
        MoveL Target_1750,v100,z10,Marcador_R\WObj:=Wo_Caja;
        MoveL Target_1760,v100,z10,Marcador_R\WObj:=Wo_Caja;
        MoveL Target_1770,v100,z10,Marcador_R\WObj:=Wo_Caja;
        MoveL Target_1780,v100,z10,Marcador_R\WObj:=Wo_Caja;
        MoveL Target_1790,v100,z10,Marcador_R\WObj:=Wo_Caja;
        MoveL Target_1800,v100,z10,Marcador_R\WObj:=Wo_Caja;
        MoveL Target_1810,v100,z10,Marcador_R\WObj:=Wo_Caja;
        MoveL Target_1820,v100,z10,Marcador_R\WObj:=Wo_Caja;
        MoveL Target_1830,v100,z10,Marcador_R\WObj:=Wo_Caja;
        MoveL Target_1840,v100,z10,Marcador_R\WObj:=Wo_Caja;
        MoveL Target_1850,v100,z10,Marcador_R\WObj:=Wo_Caja;
        MoveL Target_1860,v100,z10,Marcador_R\WObj:=Wo_Caja;
        MoveL Target_1870,v100,z10,Marcador_R\WObj:=Wo_Caja;
        MoveL Target_1880,v100,z10,Marcador_R\WObj:=Wo_Caja;
        MoveL Target_1890,v100,z10,Marcador_R\WObj:=Wo_Caja;
        MoveL Target_1900,v100,z10,Marcador_R\WObj:=Wo_Caja;
        MoveL Target_1910,v100,z10,Marcador_R\WObj:=Wo_Caja;
        MoveL Target_1920,v100,z10,Marcador_R\WObj:=Wo_Caja;
    ENDPROC

    PROC Path_30()
        MoveJ Target_Home,v100,z10,tool0\WObj:=wobj0;
    ENDPROC
    PROC Path_40()
        MoveJ Target_1930,v100,z10,Marcador_R\WObj:=Wo_Caja;
        MoveL Target_1940,v100,z10,Marcador_R\WObj:=Wo_Caja;
        MoveL Target_1950,v100,z10,Marcador_R\WObj:=Wo_Caja;
        MoveL Target_1960,v100,z10,Marcador_R\WObj:=Wo_Caja;
        MoveL Target_1970,v100,z10,Marcador_R\WObj:=Wo_Caja;
        MoveL Target_1980,v100,z10,Marcador_R\WObj:=Wo_Caja;
        MoveL Target_1990,v100,z10,Marcador_R\WObj:=Wo_Caja;
        MoveL Target_2000,v100,z10,Marcador_R\WObj:=Wo_Caja;
        MoveL Target_2010,v100,z10,Marcador_R\WObj:=Wo_Caja;
        MoveL Target_2020,v100,z10,Marcador_R\WObj:=Wo_Caja;
        MoveL Target_1930,v100,z10,Marcador_R\WObj:=Wo_Caja;
        MoveL Target_2040,v100,z10,Marcador_R\WObj:=Wo_Caja;
    ENDPROC
    PROC Path_50()
        MoveJ Target_2060,v100,z10,tool0\WObj:=wobj0;
    ENDPROC
ENDMODULE
